# EPICS StreamDevice protocol: protocols/wr.proto
Terminator = LF;
ExtraInput = Ignore;

getCount {
	out "\$1";
	in "%d";
}

getTaiDate {
	out "tai_date";
	in "%#s";
}

getSi5326TP_STATE {
	out "si5326_tune_phase.state";
	in "%#s";
}

getSi5326TP_STATE_VALUE {
	in "%*d %s %*d %*s";
}

getSi5326TP_OK {
	in "%*d %*s %*d %*s %*d %d";
}

getSi5326TP_BUSY {
	in "%*d %*s %*d %*s %d %*d";
}

setSi5326TP {
	out "si5326_tune_phase 1";
	in "";
}
